KUKA KRL program: caja_g_m3.src, caja_g_m3.dat

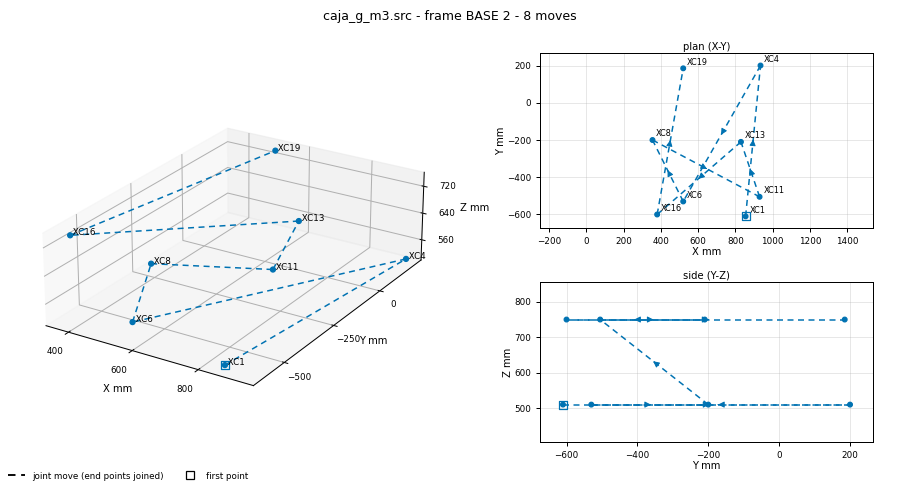
[picture p0: tool path of caja_g_m3.src in frame BASE 2, 8 of 19 moves have a stored position in this frame; points joined in program order, loops and branches not executed]
--- caja_g_m3.src ---
&ACCESS RVO1
&REL 23
&PARAM DISKPATH = KRC:\R1\Program\CAJA_G
&PARAM TEMPLATE = C:\KRC\Roboter\Template\vorgabe
&PARAM EDITMASK = *
DEF caja_g_m3( )
;Fold DECLARACION VARIABLES
DECL E6POS POS_0
DECL E6POS POS_A
DECL E6POS POS_B
DECL E6POS POS_C
DECL E6POS POS_D
DECL INT PLANTA
DECL INT SACOS_A_PALETIZAR
DECL E6POS PUNTO[20]
DECL INT n
DECL REAL INC_Z
EXT COGE_G()
;Endfold
;FOLD INI;%{PE}
  ;FOLD BASISTECH INI
    GLOBAL INTERRUPT DECL 3 WHEN $STOPMESS==TRUE DO IR_STOPM ( )
    INTERRUPT ON 3
    BAS (#INITMOV,0 )
  ;ENDFOLD (BASISTECH INI)
;FOLD SPOTTECH INI
USERSPOT(#INIT)
;ENDFOLD (SPOTTECH INI)
;FOLD GRIPPERTECH INI
USER_GRP(0,DUMMY,DUMMY,GDEFAULT)
;ENDFOLD (GRIPPERTECH INI)
  ;FOLD USER INI
    ;Make your modifications here

  ;ENDFOLD (USER INI)
;ENDFOLD (INI)
; === PROGRAMA PALETIZADO CAJAS CYREN 2x10 Kg ==
;Fold VARIABLES
PLANTA = 1
N_SACO=0
SACOS_A_PALETIZAR=SACOS_REALZIAR
n=1
INC_Z=5   ;Cota Inicial Dejada
PUNTO[1]=XC1
PUNTO[2]=XC2
PUNTO[3]=XC3
PUNTO[4]=XC4
PUNTO[5]=XC5
PUNTO[6]=XC6
PUNTO[7]=XC7
PUNTO[8]=XC8
PUNTO[9]=XC9
PUNTO[10]=XC10
PUNTO[11]=XC11
PUNTO[12]=XC12
PUNTO[13]=XC13
PUNTO[14]=XC14
PUNTO[15]=XC15
PUNTO[16]=XC16
PUNTO[17]=XC17
PUNTO[18]=XC18
PUNTO[19]=XC19
PUNTO[20]=XC20
;Endfold
;FOLD PTP HOME1  Vel= 100 % DEFAULT;%{PE}%MKUKATPBASIS,%CMOVE,%VPTP,%P 1:PTP, 2:HOME1, 3:, 5:100, 7:DEFAULT
$BWDSTART = FALSE
PDAT_ACT=PDEFAULT
FDAT_ACT=FHOME
BAS (#PTP_PARAMS,100 )
$H_POS=XHOME1
PTP  XHOME1
;ENDFOLD
;Fold Compruebo Palet
WAIT FOR PALET_LIBRE OR SALIR_PROGRAMA_ACTUAL
IF SALIR_PROGRAMA_ACTUAL == TRUE THEN
   PULSE ( OK_LEIDO_SALIR_PROGRAMA, true, 0.5 )
   WAIT SEC 1
   GOTO SALIRPROG
ENDIF
;Endfold

BOMBA =TRUE
;=== BUCLE PRINCIPAL ==
FOR PLANTA=1 TO 5 ;Bucle de plantas
FOR n=1 TO 20 ;Bucle de cajas
CAJA:

;Fold Espero señal PLC:  REPITE_CAJA
IF (ERROR_SACO_CAIDO == TRUE ) THEN
   WAIT FOR REPITE_SACO OR SALIR_PROGRAMA_ACTUAL
   ERROR_SACO_CAIDO = FALSE

   IF SALIR_PROGRAMA_ACTUAL == TRUE THEN
   PULSE ( OK_LEIDO_SALIR_PROGRAMA, true, 0.5 )
   WAIT SEC 1
   GOTO SALIRPROG
   ENDIF

ENDIF
;Endfold
COGE_G () ;Llamo programa coger
;Fold CONDICION DE SALIDA DE PROGRAMA PLC
IF SALIR == TRUE THEN
   GOTO SALIRPROG
ENDIF
;Endfold

BAS(#BASE,2) ;Cambio de base
$APO.CPTP = 70

;Fold DEFINICION PUNTOS AUXILIARES
POS_0 =PUNTO[n]
POS_A =PUNTO[n]
POS_B =PUNTO[n]
POS_C =PUNTO[n]
POS_D =PUNTO[n]

POS_0.Y=POS_0.Y+80
POS_0.X=POS_0.X-80
POS_0.Z=POS_0.Z+INC_Z+700

POS_A.Y=POS_A.Y+80
POS_A.X=POS_A.X-80
POS_A.Z=POS_A.Z+INC_Z+300

POS_B.Z=POS_B.Z+INC_Z+60

POS_C.Z=POS_C.Z+INC_Z

POS_D.Z=POS_D.Z+INC_Z+300


;Endfold

;Fold Velocidad CAJA GRANDE
FOR ax_num=1 TO 6
$VEL_AXIS[ax_num]=vptpCAJAG
$ACC_AXIS[ax_num]=vaccCAJAG
ENDFOR
$VEL.CP=vlinCAJAG
;Endfold

PTP POS_0 C_PTP
PTP POS_A C_PTP

;Fold Velocidad Lenta
FOR ax_num=1 TO 6
$VEL_AXIS[ax_num]=vptpL
$ACC_AXIS[ax_num]=vaccL
ENDFOR
$VEL.CP=vlinL
;Endfold

LIN POS_B C_DIS
LIN POS_C

;Fold Compruebo caida de CAJA
IF (VACOESTATO == FALSE) THEN ;Condicion de saco perdido
   ERROR_SACO_CAIDO = TRUE
   FOR ax_num=1 TO 6
   $VEL_AXIS[ax_num]=vptpR
   $ACC_AXIS[ax_num]=vaccR
   ENDFOR
   $VEL.CP=vlinR
   LIN POS_A
   PTP POS_0 C_PTP
   ;FOLD PTP HOME  Vel= 100 % DEFAULT;%{PE}%MKUKATPBASIS,%CMOVE,%VPTP,%P 1:PTP, 2:HOME, 3:, 5:100, 7:DEFAULT
$BWDSTART = FALSE
PDAT_ACT=PDEFAULT
FDAT_ACT=FHOME
BAS (#PTP_PARAMS,100 )
$H_POS=XHOME
PTP  XHOME
;ENDFOLD
   GOTO CAJA
ENDIF
;Endfold
;Fold Abro vacio y compruebo
WAIT SEC 0.2
VACIO=FALSE  ;Abro vacio
WAIT FOR NOT VACOESTATO ;Espero Vacoestato
;Endfold
;Fold Velocidad Rapida
Continue
FOR ax_num=1 TO 6
$VEL_AXIS[ax_num]=vptpR
$ACC_AXIS[ax_num]=vaccR
ENDFOR
$VEL.CP=vlinR
;Endfold
PTP POS_D C_PTP
PTP POS_0 C_PTP

;Fold Incremento CAJA
N_SACO=N_SACO+1
IF (N_SACO >= SACOS_A_PALETIZAR) THEN
   GOTO FINAL
ENDIF
;Endfold
ENDFOR
;Fold Incremento Planta
PLANTA = PLANTA + 1
INC_Z=INC_Z+500.0  ;Incremento cota superior
;Endfold
ENDFOR

GOTO FINAL
; Fold PUNTOS CAJAS
;FOLD PTP C1 Vel=50 % PDAT1 Tool[1]:VENTOSA_SACOS Base[2]:PALETS;%{PE}%R 8.2.24,%MKUKATPBASIS,%CMOVE,%VPTP,%P 1:PTP, 2:C1, 3:, 5:50, 7:PDAT1
$BWDSTART=FALSE
PDAT_ACT=PPDAT1
FDAT_ACT=FC1
BAS(#PTP_PARAMS,50)
PTP XC1
;ENDFOLD
;FOLD PTP C4 Vel=50 % PDAT4 Tool[1]:VENTOSA_SACOS Base[2]:PALETS;%{PE}%R 8.2.24,%MKUKATPBASIS,%CMOVE,%VPTP,%P 1:PTP, 2:C4, 3:, 5:50, 7:PDAT4
$BWDSTART=FALSE
PDAT_ACT=PPDAT4
FDAT_ACT=FC4
BAS(#PTP_PARAMS,50)
PTP XC4
;ENDFOLD
;FOLD PTP C6 Vel=50 % PDAT6 Tool[1]:VENTOSA_SACOS Base[2]:PALETS;%{PE}%R 8.2.24,%MKUKATPBASIS,%CMOVE,%VPTP,%P 1:PTP, 2:C6, 3:, 5:50, 7:PDAT6
$BWDSTART=FALSE
PDAT_ACT=PPDAT6
FDAT_ACT=FC6
BAS(#PTP_PARAMS,50)
PTP XC6
;ENDFOLD
;FOLD PTP C8 Vel=50 % PDAT8 Tool[1]:VENTOSA_SACOS Base[2]:PALETS;%{PE}%R 8.2.24,%MKUKATPBASIS,%CMOVE,%VPTP,%P 1:PTP, 2:C8, 3:, 5:50, 7:PDAT8
$BWDSTART=FALSE
PDAT_ACT=PPDAT8
FDAT_ACT=FC8
BAS(#PTP_PARAMS,50)
PTP XC8
;ENDFOLD

;Planta 2
;FOLD PTP C11 Vel=50 % PDAT11 Tool[1]:VENTOSA_SACOS Base[2]:PALETS;%{PE}%R 8.2.24,%MKUKATPBASIS,%CMOVE,%VPTP,%P 1:PTP, 2:C11, 3:, 5:50, 7:PDAT11
$BWDSTART=FALSE
PDAT_ACT=PPDAT11
FDAT_ACT=FC11
BAS(#PTP_PARAMS,50)
PTP XC11
;ENDFOLD
;FOLD PTP C13 Vel=50 % PDAT13 Tool[1]:VENTOSA_SACOS Base[2]:PALETS;%{PE}%R 8.2.24,%MKUKATPBASIS,%CMOVE,%VPTP,%P 1:PTP, 2:C13, 3:, 5:50, 7:PDAT13
$BWDSTART=FALSE
PDAT_ACT=PPDAT13
FDAT_ACT=FC13
BAS(#PTP_PARAMS,50)
PTP XC13
;ENDFOLD
;FOLD PTP C16 Vel=50 % PDAT16 Tool[1]:VENTOSA_SACOS Base[2]:PALETS;%{PE}%R 8.2.24,%MKUKATPBASIS,%CMOVE,%VPTP,%P 1:PTP, 2:C16, 3:, 5:50, 7:PDAT16
$BWDSTART=FALSE
PDAT_ACT=PPDAT16
FDAT_ACT=FC16
BAS(#PTP_PARAMS,50)
PTP XC16
;ENDFOLD
;FOLD PTP C19 Vel=50 % PDAT19 Tool[1]:VENTOSA_SACOS Base[2]:PALETS;%{PE}%R 8.2.24,%MKUKATPBASIS,%CMOVE,%VPTP,%P 1:PTP, 2:C19, 3:, 5:50, 7:PDAT19
$BWDSTART=FALSE
PDAT_ACT=PPDAT19
FDAT_ACT=FC19
BAS(#PTP_PARAMS,50)
PTP XC19
;ENDFOLD

;Endfold


FINAL:

PULSE ( PALET_COMPLETO, TRUE, 0.5 )
WAIT SEC 1

SALIRPROG:

N_SACO=0
SALIR=FALSE
BOMBA=FALSE

;FOLD PTP HOME CONT Vel=ptpM % DEFAULT;%{PE}%R 8.2.24,%MKUKATPBASIS,%CMOVE,%VPTP,%P 1:PTP, 2:HOME, 3:C_DIS, 5:50, 7:DEFAULT
$BWDSTART=FALSE
PDAT_ACT=PDEFAULT
FDAT_ACT=FHOME
BAS(#PTP_PARAMS,vptpM)
$H_POS=XHOME
$APO.CPTP = 70
PTP XHOME C_PTP
;ENDFOLD

END

--- caja_g_m3.dat ---
&ACCESS RVO1
&REL 23
&PARAM DISKPATH = KRC:\R1\Program\CAJA_G
&PARAM TEMPLATE = C:\KRC\Roboter\Template\vorgabe
&PARAM EDITMASK = *
DEFDAT  caja_g_m3
;FOLD EXTERNAL DECLARATIONS;%{PE}%MKUKATPBASIS,%CEXT,%VCOMMON,%P
;FOLD GRIPPERTECH EXT
EXT  H50 (INT  :IN,INT  :IN,INT  :IN,GRP_TYP  :IN )
;ENDFOLD (GRIPPERTECH EXT)
;FOLD SPOTTECH EXT
EXT  USERSPOT (S_COMMAND  :IN,SPOT_TYPE  :IN )
;ENDFOLD (SPOTTECH EXT)
;FOLD BASISTECH EXT;%{PE}%MKUKATPBASIS,%CEXT,%VEXT,%P
EXT  BAS (BAS_COMMAND  :IN,REAL  :IN )
DECL INT SUCCESS
;ENDFOLD (BASISTECH EXT)
;FOLD USER EXT;%{E}%MKUKATPUSER,%CEXT,%VEXT,%P
;Make your modifications here

;ENDFOLD (USER EXT)
;ENDFOLD (EXTERNAL DECLARATIONS)
DECL BASIS_SUGG_T LAST_BASIS={POINT1[] "C19                     ",POINT2[] "C19                     ",CP_PARAMS[] "CPDAT0                  ",PTP_PARAMS[] "PDAT19                  ",CONT[] "                        ",CP_VEL[] "2.0                     ",PTP_VEL[] "50                      ",SYNC_PARAMS[] "SYNCDAT                 ",SPL_NAME[] "S0                      "}

DECL E6POS XC1={X 855.0,Y -610.0,Z 510.0,A 85.683197,B 0.372132391,C -179.818298,S 2,T 43,E1 0.0,E2 0.0,E3 0.0,E4 0.0,E5 0.0,E6 0.0}
DECL FDAT FC1={TOOL_NO 1,BASE_NO 2,IPO_FRAME #BASE,POINT2[] " ",TQ_STATE FALSE}
DECL PDAT PPDAT1={VEL 100.0,ACC 100.0,APO_DIST 100.0,APO_MODE #CDIS,GEAR_JERK 50.0}
DECL E6POS XC2={X 855.0,Y -370.0,Z 510.0,A 85.683197,B 0.372132391,C -179.818298,S 2,T 43,E1 0.0,E2 0.0,E3 0.0,E4 0.0,E5 0.0,E6 0.0}
DECL FDAT FC2={TOOL_NO 1,BASE_NO 2,IPO_FRAME #BASE,POINT2[] " ",TQ_STATE FALSE}
DECL PDAT PPDAT2={VEL 100.0,ACC 100.0,APO_DIST 100.0,APO_MODE #CDIS,GEAR_JERK 50.0}
DECL E6POS XC3={X 855.0,Y -130.0,Z 510.0,A 85.683197,B 0.372132391,C -179.818298,S 2,T 43,E1 0.0,E2 0.0,E3 0.0,E4 0.0,E5 0.0,E6 0.0}
DECL FDAT FC3={TOOL_NO 1,BASE_NO 2,IPO_FRAME #BASE,POINT2[] " ",TQ_STATE FALSE}
DECL PDAT PPDAT3={VEL 100.0,ACC 100.0,APO_DIST 100.0,APO_MODE #CDIS,GEAR_JERK 50.0}

DECL E6POS XC4={X 935.0,Y 200.0,Z 510.0,A 174.968307,B -0.174836293,C -179.624603,S 2,T 11,E1 0.0,E2 0.0,E3 0.0,E4 0.0,E5 0.0,E6 0.0}
DECL FDAT FC4={TOOL_NO 1,BASE_NO 2,IPO_FRAME #BASE,POINT2[] " ",TQ_STATE FALSE}
DECL PDAT PPDAT4={VEL 100.0,ACC 100.0,APO_DIST 100.0,APO_MODE #CDIS,GEAR_JERK 50.0}
DECL E6POS XC5={X 695.0,Y 200.0,Z 510.0,A 174.968307,B -0.174836293,C -179.624603,S 2,T 11,E1 0.0,E2 0.0,E3 0.0,E4 0.0,E5 0.0,E6 0.0}
DECL FDAT FC5={TOOL_NO 1,BASE_NO 2,IPO_FRAME #BASE,POINT2[] " ",TQ_STATE FALSE}
DECL PDAT PPDAT5={VEL 100.0,ACC 100.0,APO_DIST 100.0,APO_MODE #CDIS,GEAR_JERK 50.0}

DECL E6POS XC6={X 520.0,Y -530.0,Z 510.0,A -2.75768495,B 0.189947397,C 179.631607,S 2,T 35,E1 0.0,E2 0.0,E3 0.0,E4 0.0,E5 0.0,E6 0.0}
DECL FDAT FC6={TOOL_NO 1,BASE_NO 2,IPO_FRAME #BASE,POINT2[] " ",TQ_STATE FALSE}
DECL PDAT PPDAT6={VEL 100.0,ACC 100.0,APO_DIST 100.0,APO_MODE #CDIS,GEAR_JERK 50.0}
DECL E6POS XC7={X 280.0,Y -530.0,Z 510.0,A -2.75768495,B 0.189947397,C 179.631607,S 2,T 35,E1 0.0,E2 0.0,E3 0.0,E4 0.0,E5 0.0,E6 0.0}
DECL FDAT FC7={TOOL_NO 1,BASE_NO 2,IPO_FRAME #BASE,POINT2[] " ",TQ_STATE FALSE}
DECL PDAT PPDAT7={VEL 100.0,ACC 100.0,APO_DIST 100.0,APO_MODE #CDIS,GEAR_JERK 50.0}

DECL E6POS XC8={X 355.0,Y -200.0,Z 510,A -92.9248734,B -0.368633211,C 179.810806,S 2,T 3,E1 0.0,E2 0.0,E3 0.0,E4 0.0,E5 0.0,E6 0.0}
DECL FDAT FC8={TOOL_NO 1,BASE_NO 2,IPO_FRAME #BASE,POINT2[] " ",TQ_STATE FALSE}
DECL PDAT PPDAT8={VEL 100.0,ACC 100.0,APO_DIST 100.0,APO_MODE #CDIS,GEAR_JERK 50.0}
DECL E6POS XC9={X 355.0,Y 40.0,Z 510,A -92.9248734,B -0.368633211,C 179.810806,S 2,T 3,E1 0.0,E2 0.0,E3 0.0,E4 0.0,E5 0.0,E6 0.0}
DECL FDAT FC9={TOOL_NO 1,BASE_NO 2,IPO_FRAME #BASE,POINT2[] " ",TQ_STATE FALSE}
DECL PDAT PPDAT9={VEL 100.0,ACC 100.0,APO_DIST 100.0,APO_MODE #CDIS,GEAR_JERK 50.0}
DECL E6POS XC10={X 355.0,Y 280.0,Z 510,A -92.9248734,B -0.368633211,C 179.810806,S 2,T 3,E1 0.0,E2 0.0,E3 0.0,E4 0.0,E5 0.0,E6 0.0}
DECL FDAT FC10={TOOL_NO 1,BASE_NO 2,IPO_FRAME #BASE,POINT2[] " ",TQ_STATE FALSE}
DECL PDAT PPDAT10={VEL 100.0,ACC 100.0,APO_DIST 100.0,APO_MODE #CDIS,GEAR_JERK 50.0}

;Planta 2

DECL E6POS XC11={X 930.0,Y -505.0,Z 750.0,A 175.158798,B -0.177922398,C -179.6259,S 2,T 11,E1 0.0,E2 0.0,E3 0.0,E4 0.0,E5 0.0,E6 0.0}
DECL FDAT FC11={TOOL_NO 1,BASE_NO 2,IPO_FRAME #BASE,POINT2[] " ",TQ_STATE FALSE}
DECL PDAT PPDAT11={VEL 100.0,ACC 100.0,APO_DIST 100.0,APO_MODE #CDIS,GEAR_JERK 50.0}
DECL E6POS XC12={X 690.0,Y -505.0,Z 750.0,A 175.158798,B -0.177922398,C -179.6259,S 2,T 11,E1 0.0,E2 0.0,E3 0.0,E4 0.0,E5 0.0,E6 0.0}
DECL FDAT FC12={TOOL_NO 1,BASE_NO 2,IPO_FRAME #BASE,POINT2[] " ",TQ_STATE FALSE}
DECL PDAT PPDAT12={VEL 100.0,ACC 100.0,APO_DIST 100.0,APO_MODE #CDIS,GEAR_JERK 50.0}

DECL E6POS XC13={X 830.0,Y -210.0,Z 750.0,A -93.0405807,B -0.36804691,C 179.809601,S 2,T 3,E1 0.0,E2 0.0,E3 0.0,E4 0.0,E5 0.0,E6 0.0}
DECL FDAT FC13={TOOL_NO 1,BASE_NO 2,IPO_FRAME #BASE,POINT2[] " ",TQ_STATE FALSE}
DECL PDAT PPDAT13={VEL 100.0,ACC 100.0,APO_DIST 100.0,APO_MODE #CDIS,GEAR_JERK 50.0}
DECL E6POS XC14={X 830.0,Y 30.0,Z 750.0,A -93.0405807,B -0.36804691,C 179.809601,S 2,T 3,E1 0.0,E2 0.0,E3 0.0,E4 0.0,E5 0.0,E6 0.0}
DECL FDAT FC14={TOOL_NO 1,BASE_NO 2,IPO_FRAME #BASE,POINT2[] " ",TQ_STATE FALSE}
DECL PDAT PPDAT14={VEL 100.0,ACC 100.0,APO_DIST 100.0,APO_MODE #CDIS,GEAR_JERK 50.0}
DECL E6POS XC15={X 830.0,Y 270.0,Z 750.0,A -93.0405807,B -0.36804691,C 179.809601,S 2,T 3,E1 0.0,E2 0.0,E3 0.0,E4 0.0,E5 0.0,E6 0.0}
DECL FDAT FC15={TOOL_NO 1,BASE_NO 2,IPO_FRAME #BASE,POINT2[] " ",TQ_STATE FALSE}
DECL PDAT PPDAT15={VEL 100.0,ACC 100.0,APO_DIST 100.0,APO_MODE #CDIS,GEAR_JERK 50.0}

DECL E6POS XC16={X 380.0,Y -600.0,Z 750.0,A 85.5915298,B 0.371447891,C -179.8181,S 2,T 43,E1 0.0,E2 0.0,E3 0.0,E4 0.0,E5 0.0,E6 0.0}
DECL FDAT FC16={TOOL_NO 1,BASE_NO 2,IPO_FRAME #BASE,POINT2[] " ",TQ_STATE FALSE}
DECL PDAT PPDAT16={VEL 100.0,ACC 100.0,APO_DIST 100.0,APO_MODE #CDIS,GEAR_JERK 50.0}
DECL E6POS XC17={X 380.0,Y -360.0,Z 750.0,A 85.5915298,B 0.371447891,C -179.8181,S 2,T 43,E1 0.0,E2 0.0,E3 0.0,E4 0.0,E5 0.0,E6 0.0}
DECL FDAT FC17={TOOL_NO 1,BASE_NO 2,IPO_FRAME #BASE,POINT2[] " ",TQ_STATE FALSE}
DECL PDAT PPDAT17={VEL 100.0,ACC 100.0,APO_DIST 100.0,APO_MODE #CDIS,GEAR_JERK 50.0}
DECL E6POS XC18={X 380.0,Y -120.0,Z 750.0,A 85.5915298,B 0.371447891,C -179.8181,S 2,T 43,E1 0.0,E2 0.0,E3 0.0,E4 0.0,E5 0.0,E6 0.0}
DECL FDAT FC18={TOOL_NO 1,BASE_NO 2,IPO_FRAME #BASE,POINT2[] " ",TQ_STATE FALSE}
DECL PDAT PPDAT18={VEL 100.0,ACC 100.0,APO_DIST 100.0,APO_MODE #CDIS,GEAR_JERK 50.0}

DECL E6POS XC19={X 520.0,Y 185.0,Z 750.0,A -5.186656,B 0.174743995,C 179.624298,S 2,T 35,E1 0.0,E2 0.0,E3 0.0,E4 0.0,E5 0.0,E6 0.0}
DECL FDAT FC19={TOOL_NO 1,BASE_NO 2,IPO_FRAME #BASE,POINT2[] " ",TQ_STATE FALSE}
DECL PDAT PPDAT19={VEL 100.0,ACC 100.0,APO_DIST 100.0,APO_MODE #CDIS,GEAR_JERK 50.0}
DECL E6POS XC20={X 280.0,Y 185.0,Z 750.0,A -5.186656,B 0.174743995,C 179.624298,S 2,T 35,E1 0.0,E2 0.0,E3 0.0,E4 0.0,E5 0.0,E6 0.0}
DECL FDAT FC20={TOOL_NO 1,BASE_NO 2,IPO_FRAME #BASE,POINT2[] " ",TQ_STATE FALSE}
DECL PDAT PPDAT20={VEL 100.0,ACC 100.0,APO_DIST 100.0,APO_MODE #CDIS,GEAR_JERK 50.0}

ENDDAT
